KUKA KRL program: coge_25.src, coge_25.dat

--- coge_25.src ---
&ACCESS RVO1
&REL 13
&PARAM TEMPLATE = C:\KRC\Roboter\Template\vorgabe
&PARAM EDITMASK = *
DEF coge_25( )
;Fold Definicion de Variables
DECL E6POS POS_AUX1
DECL REAL INC_Z1
;Endfold
;FOLD INI;%{PE}
  ;FOLD BASISTECH INI
    GLOBAL INTERRUPT DECL 3 WHEN $STOPMESS==TRUE DO IR_STOPM ( )
    INTERRUPT ON 3
    BAS (#INITMOV,0 )
  ;ENDFOLD (BASISTECH INI)
;FOLD SPOTTECH INI
USERSPOT(#INIT)
;ENDFOLD (SPOTTECH INI)
;FOLD GRIPPERTECH INI
USER_GRP(0,DUMMY,DUMMY,GDEFAULT)
;ENDFOLD (GRIPPERTECH INI)
  ;FOLD USER INI
    ;Make your modifications here

  ;ENDFOLD (USER INI)
;ENDFOLD (INI)
; === PROGRAMA COGIDA SACOS 20 KG ==
;Fold VARIABLES
INC_Z1=350 ;Cota Inicial Seguridad 350
POS_AUX1 =XC1
POS_AUX1.Z=POS_AUX1.Z+INC_Z1
;Endfold

;FOLD PTP HOME CONT Vel=100 % DEFAULT;%{PE}%R 8.2.24,%MKUKATPBASIS,%CMOVE,%VPTP,%P 1:PTP, 2:HOME, 3:C_DIS, 5:50, 7:DEFAULT
$BWDSTART=FALSE
PDAT_ACT=PDEFAULT
FDAT_ACT=FHOME
BAS(#PTP_PARAMS,100)
$H_POS=XHOME
PTP XHOME C_DIS
;ENDFOLD

$ADVANCE=2
BAS(#BASE,1)

;Fold Cambio velocidad Rapida
Continue
FOR ax_num=1 TO 6
$VEL_AXIS[ax_num]=vptpR
$ACC_AXIS[ax_num]=vaccR
ENDFOR
$VEL.CP=vlinR
;Endfold

PTP POS_AUX1 C_DIS

;Fold Espero señal PLC: Saco RDY
WAIT FOR SACO_RDY OR SALIR_PROGRAMA_ACTUAL
IF SALIR_PROGRAMA_ACTUAL == TRUE THEN
   PULSE ( OK_LEIDO_SALIR_PROGRAMA, true, 0.5 )
   SALIR = TRUE
   WAIT SEC 1
   GOTO FINAL
ENDIF
;Endfold

VACIO=TRUE ;Cierro vacio
LIN XC1 ;Punto Cogida Saco
WAIT FOR VACOESTATO OR SALIR_PROGRAMA_ACTUAL OR VOLVER_COGER;Espero Vacoestato

;Fold Cambio velocidad Media
$VEL.CP=vlinM
;Endfold
LIN POS_AUX1 C_DIS

CONTINUE
PULSE ( SACO_COGIDO, TRUE, 0.5 ) ;Indico saco cogido
;FOLD PTP HOME CONT Vel=ptpM % DEFAULT;%{PE}%R 8.2.24,%MKUKATPBASIS,%CMOVE,%VPTP,%P 1:PTP, 2:HOME, 3:C_DIS, 5:50, 7:DEFAULT
$BWDSTART=FALSE
PDAT_ACT=PDEFAULT
FDAT_ACT=FHOME
BAS(#PTP_PARAMS,vptpM)
$H_POS=XHOME
$APO.CPTP = 70
PTP XHOME C_PTP
;ENDFOLD

;PUNTOS COGIDA SOLO PARA MODIFICAR TOUCHAP
GOTO FINAL
;FOLD PTP C1 Vel=100 % PDAT2 Tool[1]:VENTOSA_SACOS Base[1]:SACOS;%{PE}%R 8.2.24,%MKUKATPBASIS,%CMOVE,%VPTP,%P 1:PTP, 2:C1, 3:, 5:100, 7:PDAT2
$BWDSTART=FALSE
PDAT_ACT=PPDAT2
FDAT_ACT=FC1
BAS(#PTP_PARAMS,100)
PTP XC1 C_DIS
;ENDFOLD
FINAL:
END

--- coge_25.dat ---
&ACCESS RVO1
&REL 13
&PARAM TEMPLATE = C:\KRC\Roboter\Template\vorgabe
&PARAM EDITMASK = *
DEFDAT  coge_25
;FOLD EXTERNAL DECLARATIONS;%{PE}%MKUKATPBASIS,%CEXT,%VCOMMON,%P
;FOLD GRIPPERTECH EXT
EXT  H50 (INT  :IN,INT  :IN,INT  :IN,GRP_TYP  :IN )
;ENDFOLD (GRIPPERTECH EXT)
;FOLD SPOTTECH EXT
EXT  USERSPOT (S_COMMAND  :IN,SPOT_TYPE  :IN )
;ENDFOLD (SPOTTECH EXT)
;FOLD BASISTECH EXT;%{PE}%MKUKATPBASIS,%CEXT,%VEXT,%P
EXT  BAS (BAS_COMMAND  :IN,REAL  :IN )
DECL INT SUCCESS
;ENDFOLD (BASISTECH EXT)
;FOLD USER EXT;%{E}%MKUKATPUSER,%CEXT,%VEXT,%P
;Make your modifications here

;ENDFOLD (USER EXT)
;ENDFOLD (EXTERNAL DECLARATIONS)
DECL BASIS_SUGG_T LAST_BASIS={POINT1[] "SALVOPRECINTADORA       ",POINT2[] "SALVOPRECINTADORA       ",CP_PARAMS[] "CPDAT1                  ",PTP_PARAMS[] "PDAT5                   ",CONT[] "C_DIS                   ",CP_VEL[] "0.4                     ",PTP_VEL[] "50                      ",SYNC_PARAMS[] "SYNCDAT                 ",SPL_NAME[] "S0                      "}
DECL E6POS XC1={X 319.906799,Y 1434.229,Z 170.114304,A 175.524399,B 0.675907314,C -179.652496,S 6,T 18,E1 0.0,E2 0.0,E3 0.0,E4 0.0,E5 0.0,E6 0.0}
DECL FDAT FC1={TOOL_NO 1,BASE_NO 1,IPO_FRAME #BASE,POINT2[] " ",TQ_STATE FALSE}
DECL PDAT PPDAT2={VEL 100.0,ACC 100.0,APO_DIST 100.0,APO_MODE #CDIS,GEAR_JERK 50.0}
ENDDAT
